// TIA Portal V20 export
DATA_BLOCK "Test"   // DB70
// stored: Access Published, MemoryReserve 100, Namespace Unit1
   VAR
      "Bool" : Array[0..999] of Bool;
      "DInt" : Array[0..9] of DInt;
      partDataA { S7_SetPoint := 'True'} : "LER_typePartData";
      partDataB { S7_SetPoint := 'True'} : "LER_typePartData";
      transfer { S7_SetPoint := 'True'} : Bool;
      detect : Bool;
      emNumber : Int;
   END_VAR
BEGIN
   // "Bool"[0] : Part Data Delete
   // "Bool"[4] : Safety realese by pass
   // "Bool"[10] : Production Mode
   // "Bool"[11] : Maintance Mode
   // "Bool"[12] : Manual Mode
   // "Bool"[20] : START
   // "Bool"[21] : STOP
   // "Bool"[22] : HOME
   // "Bool"[23] : RESET
   // "Bool"[90] : 3rd Press OK
   // "Bool"[91] : 3rd Press NG
   // "Bool"[92] : Thickness OK
   // "Bool"[93] : Thickness NG
   // "Bool"[94] : Hipot OK
   // "Bool"[95] : Hipot NG
   // "Bool"[96] : Vision OK
   // "Bool"[97] : Vision NG
   // "Bool"[98] : QR Read OK
   // "Bool"[99] : QR Read NG
   // "Bool"[100] : QR Data Compare OK
   // "Bool"[101] : QR Data Compare NG
END_DATA_BLOCK
